TYPE DigitalOutputBase_1FE0D5EE :
STRUCT
END_STRUCT
END_TYPE

(* stored: Version 1.2.0.0, ProductVersion 3.1.4024.9
   DUT DigitalOutputBase_1FE0D5EE: Id {41d2aa2c-c179-416c-9efc-097a23176cf3} *)
